Fanuc KAREL source: kf00099.KL

-- PROVISIONAL review KL for V770-1; original PC SHA256 b2fb8fcac37217dd62e4cb7bf4e90028c934aadcd7540e9819bcbd9592b1005d
-- Incomplete behavior may be omitted. Consult companion uncertainty JSON. Do not deploy.
PROGRAM KF00099
%NOLOCKGROUP
BEGIN
  -- UNRESOLVED_PC offsets 5-16; opcodes 2E,23
  -- UNRESOLVED_PC offsets 21-32; opcodes 2E,23
  -- UNRESOLVED_PC offsets 37-63; opcodes 27,27,9D,22,27,9D,31,7E,4A
  -- UNRESOLVED_PC offsets 68-72; opcodes 7F
END KF00099
